// Mitsubishi GX Works2 project: PLC_Group22   PLC: FX3G

// global labels: Global1
VAR_GLOBAL
  START_DAY AT X007 : BOOL;
  EMERGENCY AT X005 : BOOL;
  DAY_IS_ON AT Y007 : BOOL;
  Input_Petel AT D2000 : REAL;
  Container_Petel AT D1100 : REAL;
  Input_Limon AT D2100 : REAL;
  Container_Limon AT D1200 : REAL;
  Input_Meyatzev AT D2200 : REAL;
  Container_Meyatzev AT D1300 : REAL;
  Input_Gumi AT D2300 : REAL;
  Container_Gumi AT D1400 : REAL;
  IceCream_Making AT X001 : BOOL;
  Gumigum_Type AT D8280 : INT;
  Chosen_Type AT D8202 : REAL;
END_VAR
VAR_GLOBAL CONSTANT
  Con_Value_6 : REAL := 6;
END_VAR
VAR_GLOBAL
  Regular AT M11 : BOOL;
  Pinuk AT M12 : BOOL;
  Enough_Petel_R AT M1 : BOOL;
  Enough_Limon_R AT M2 : BOOL;
  Enough_Meyatzev_R AT M3 : BOOL;
  Enough_Gumi_R AT M4 : BOOL;
  Enough_Regular AT M5 : BOOL;
END_VAR
VAR_GLOBAL CONSTANT
  Min_Petel_R : REAL := 280;
  Min_Limon_R : REAL := 455;
  Min_Meyatzev_R : REAL := 105;
  Min_Gumi_R : REAL := 28;
  Min_Petel_P : REAL := 385;
  Min_Limon_P : REAL := 665;
  Min_Meyatzev_P : REAL := 210;
  Min_Gumi_P : REAL := 70;
END_VAR
VAR_GLOBAL
  Enough_Petel_P AT M6 : BOOL;
  Enough_Limon_P AT M7 : BOOL;
  Enough_Meyatzev_P AT M8 : BOOL;
  Enough_Gumi_P AT M9 : BOOL;
  Enough_Pinuk AT M10 : BOOL;
END_VAR
VAR_GLOBAL CONSTANT
  Divv : REAL := 400;
  Sub280 : REAL := 280;
  Sub35 : REAL := 35;
  Sub420 : REAL := 420;
  Sub70 : REAL := 70;
  Timer5 : INT := 50;
END_VAR
VAR_GLOBAL
  IceCream_Making_Time AT TC1 : BOOL;
  StartMaking AT TS1 : BOOL;
  IsMakingIceCrem AT Y000 : BOOL;
END_VAR
VAR_GLOBAL CONSTANT
  Sub385 : REAL := 385;
  Sub105 : REAL := 105;
  Sub560 : REAL := 560;
  Sub140 : REAL := 140;
END_VAR
VAR_GLOBAL
  IceCream_Cooling AT X002 : BOOL;
END_VAR
VAR_GLOBAL CONSTANT
  Petel350 : REAL := 350;
END_VAR
VAR_GLOBAL
  CoolingPetel AT D1500 : REAL;
END_VAR
VAR_GLOBAL CONSTANT
  Limon490 : REAL := 490;
END_VAR
VAR_GLOBAL
  CoolingLimon AT D1600 : REAL;
  StartCooling AT TS2 : BOOL;
  Under10 AT X003 : BOOL;
  CoolingTimer AT TC2 : BOOL;
END_VAR
VAR_GLOBAL CONSTANT
  CoolingTime : INT := 80;
END_VAR
VAR_GLOBAL
  IsCoolingg AT Y002 : BOOL;
END_VAR
VAR_GLOBAL CONSTANT
  Petel560 : REAL := 560;
  Limon700 : REAL := 700;
END_VAR
VAR_GLOBAL
  End_Cooling_R AT M63 : BOOL;
  End_Cooling_P AT M64 : BOOL;
END_VAR
VAR_GLOBAL CONSTANT
  Cooling_Containers_R : REAL := 868;
  Gumi_R28 : REAL := 28;
END_VAR
VAR_GLOBAL
  Mixing_R_Timer AT TC3 : BOOL;
END_VAR
VAR_GLOBAL CONSTANT
  Mixing_R_Time : INT := 30;
END_VAR
VAR_GLOBAL
  Start_Mixing_R AT TS3 : BOOL;
  End_Mixing_R AT M65 : BOOL;
  Lights1 AT TC4 : BOOL;
END_VAR
VAR_GLOBAL CONSTANT
  Lights_Timer : INT := 5;
END_VAR
VAR_GLOBAL
  Lights1_on AT TS4 : BOOL;
  Lights1_Is_On AT Y005 : BOOL;
  Lights2 AT TC5 : BOOL;
  Lights2_on AT TS5 : BOOL;
  Lights2_Is_On AT Y006 : BOOL;
  Lights12 AT M66 : BOOL;
END_VAR
VAR_GLOBAL CONSTANT
  Cooling_Containers_P : REAL := 1330;
  Gumi_P70 : REAL := 70;
END_VAR
VAR_GLOBAL
  Mixing_P_Timer AT TC6 : BOOL;
END_VAR
VAR_GLOBAL CONSTANT
  Mixing_P_Time : INT := 50;
END_VAR
VAR_GLOBAL
  Start_Mixing_P AT TS6 : BOOL;
  End_Mixing_P AT M67 : BOOL;
  IceCream_Packing AT X004 : BOOL;
  Single_Unit_Packing AT X000 : BOOL;
  Units_Conter AT CC1 : BOOL;
END_VAR
VAR_GLOBAL CONSTANT
  Con_1 : REAL := 1;
END_VAR
VAR_GLOBAL
  Packages_Count AT D1900 : REAL;
  Counter_State AT CS1 : BOOL;
END_VAR
VAR_GLOBAL CONSTANT
  Min_1 : INT := 1;
  Value_7 : INT := 7;
END_VAR
VAR_GLOBAL
  Units AT CN1 : INT;
  In_Packing AT Y004 : BOOL;
  Mixing AT D1700 : REAL;
END_VAR
VAR_GLOBAL CONSTANT
  Sub124 : REAL := 124;
  Sub190 : REAL := 190;
  zero : REAL;
END_VAR
VAR_GLOBAL
  End_Packing AT M80 : BOOL;
  End_Of_The_Day AT M27 : BOOL;
  Output AT D8282 : INT;
END_VAR
VAR_GLOBAL CONSTANT
  Div40 : REAL := 40;
END_VAR
VAR_GLOBAL
  Not_Enough_Material AT M25 : BOOL;
END_VAR

// task Task_01 (event TRUE, interval 0, priority 31): POU_01

PROGRAM POU_01
(* structured ladder/FBD written out as ST: instructions are called as NAME(EN, inputs, outputs); _pN, _eN, _tN stand for wires *)
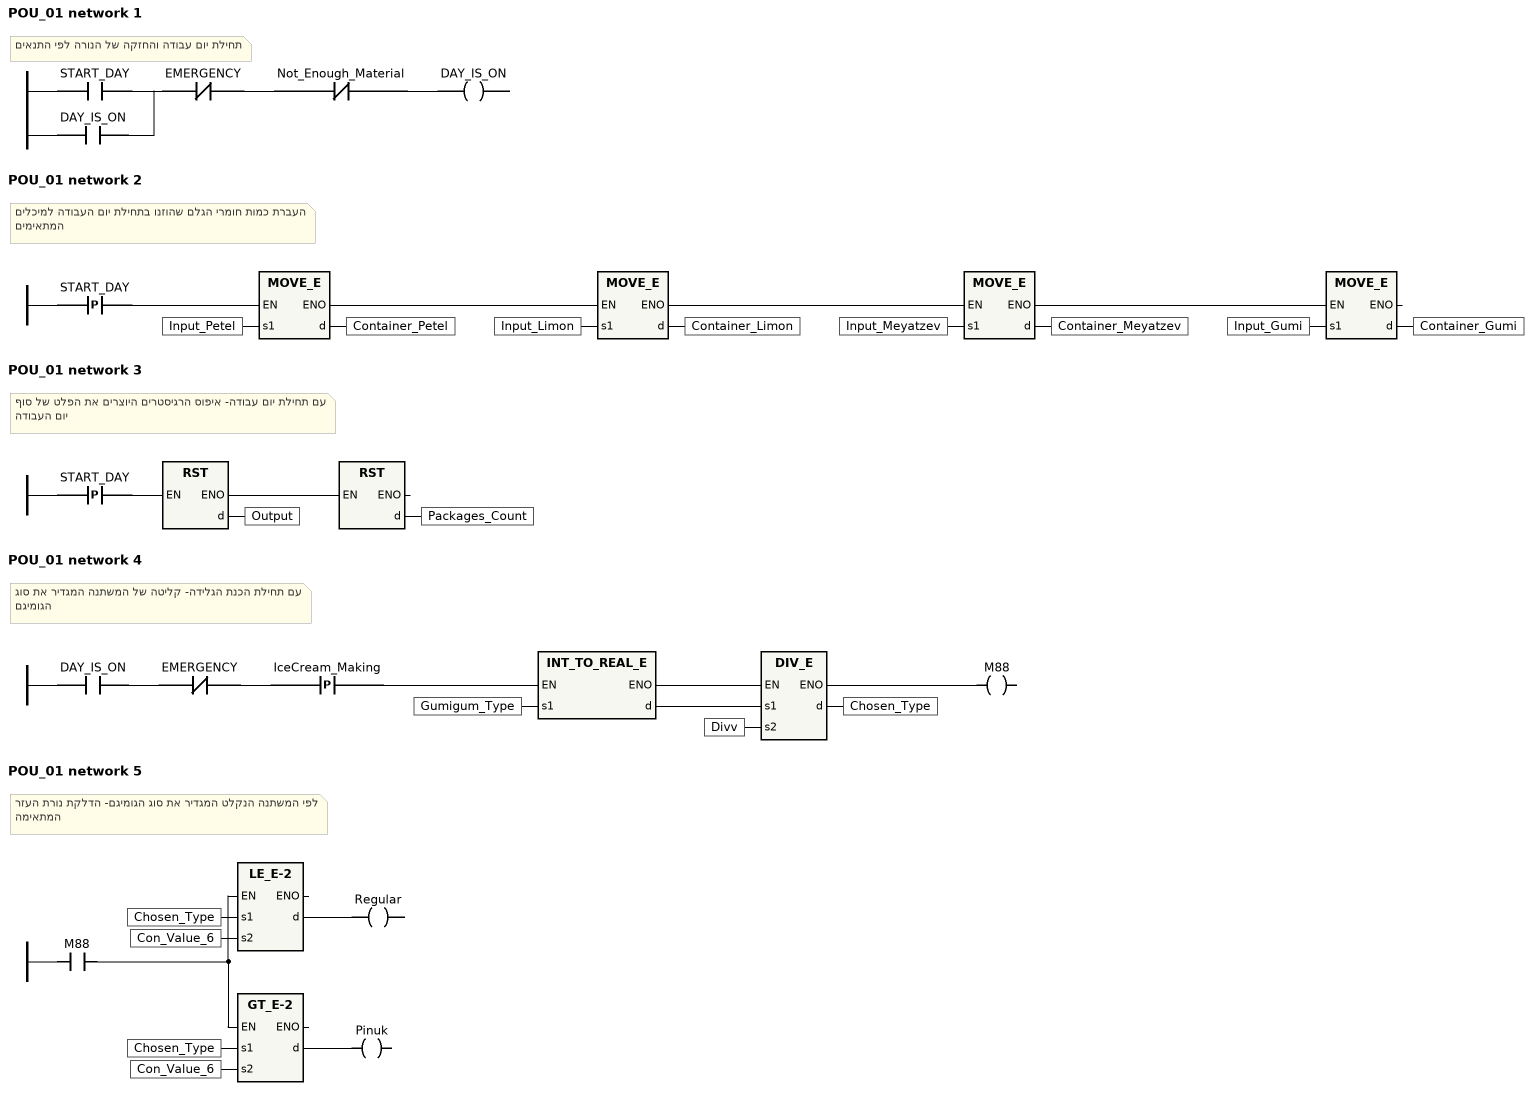
(* network 1 *)
(* תחילת יום עבודה והחזקה של הנורה לפי התנאים *)
DAY_IS_ON := ((START_DAY OR DAY_IS_ON) AND NOT EMERGENCY) AND NOT Not_Enough_Material;
(* network 2 *)
(* העברת כמות חומרי הגלם שהוזנו בתחילת יום העבודה למיכלים המתאימים *)
_e1 := MOVE_E(LDP(TRUE, START_DAY), Input_Petel, Container_Petel);
_e2 := MOVE_E(_e1, Input_Limon, Container_Limon);
_e3 := MOVE_E(_e2, Input_Meyatzev, Container_Meyatzev);
MOVE_E(_e3, Input_Gumi, Container_Gumi);
(* network 3 *)
(* עם תחילת יום עבודה- איפוס הרגיסטרים היוצרים את הפלט של סוף יום העבודה *)
_e1 := RST(LDP(TRUE, START_DAY), Output);
RST(_e1, Packages_Count);
(* network 4 *)
(* עם תחילת הכנת הגלידה- קליטה של המשתנה המגדיר את סוג הגומיגם *)
_e2 := INT_TO_REAL_E(DAY_IS_ON AND NOT EMERGENCY AND LDP(TRUE, IceCream_Making), Gumigum_Type, _t1);
_e3 := DIV_E(_e2, _t1, Divv, Chosen_Type);
M88 := _e3;
(* network 5 *)
(* לפי המשתנה הנקלט המגדיר את סוג הגומיגם- הדלקת נורת העזר המתאימה *)
LE_E(M88, Chosen_Type, Con_Value_6, _t1);
Regular := _t1;
GT_E(M88, Chosen_Type, Con_Value_6, _t2);
Pinuk := _t2;
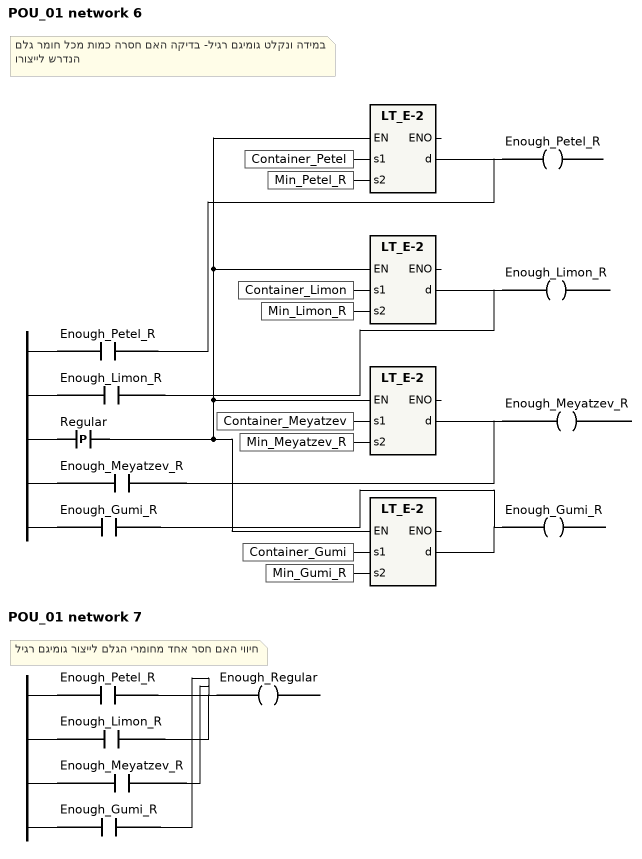
(* network 6 *)
(* במידה ונקלט גומיגם רגיל- בדיקה האם חסרה כמות מכל חומר גלם הנדרש לייצורו *)
_p1 := LDP(TRUE, Regular);
LT_E(_p1, Container_Petel, Min_Petel_R, _t2);
Enough_Petel_R := Enough_Petel_R OR _t2;
LT_E(_p1, Container_Limon, Min_Limon_R, _t3);
Enough_Limon_R := Enough_Limon_R OR _t3;
LT_E(_p1, Container_Meyatzev, Min_Meyatzev_R, _t4);
Enough_Meyatzev_R := _t4 OR Enough_Meyatzev_R;
LT_E(_p1, Container_Gumi, Min_Gumi_R, _t5);
Enough_Gumi_R := _t5 OR Enough_Gumi_R;
(* network 7 *)
(* חיווי האם חסר אחד מחומרי הגלם לייצור גומיגם רגיל *)
Enough_Regular := Enough_Petel_R OR Enough_Limon_R OR Enough_Meyatzev_R OR Enough_Gumi_R;
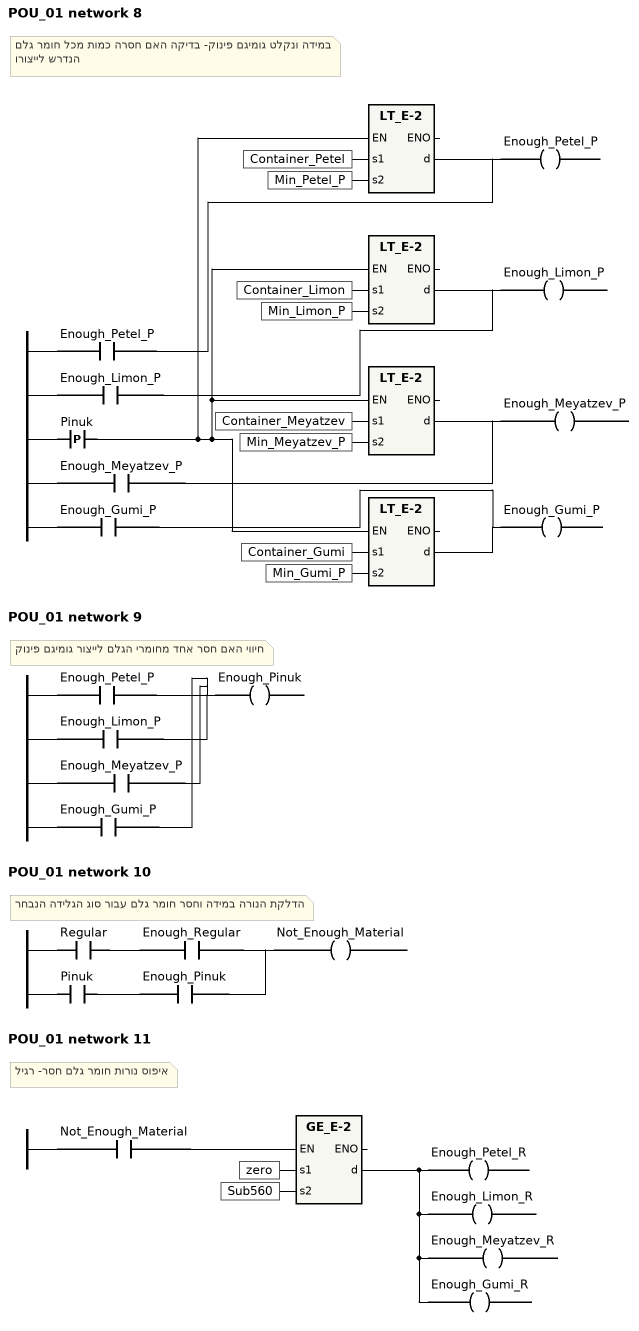
(* network 8 *)
(* במידה ונקלט גומיגם פינוק- בדיקה האם חסרה כמות מכל חומר גלם הנדרש לייצורו *)
_p1 := LDP(TRUE, Pinuk);
LT_E(_p1, Container_Petel, Min_Petel_P, _t2);
Enough_Petel_P := Enough_Petel_P OR _t2;
LT_E(_p1, Container_Limon, Min_Limon_P, _t3);
Enough_Limon_P := Enough_Limon_P OR _t3;
LT_E(_p1, Container_Meyatzev, Min_Meyatzev_P, _t4);
Enough_Meyatzev_P := _t4 OR Enough_Meyatzev_P;
LT_E(_p1, Container_Gumi, Min_Gumi_P, _t5);
Enough_Gumi_P := _t5 OR Enough_Gumi_P;
(* network 9 *)
(* חיווי האם חסר אחד מחומרי הגלם לייצור גומיגם פינוק *)
Enough_Pinuk := Enough_Petel_P OR Enough_Limon_P OR Enough_Meyatzev_P OR Enough_Gumi_P;
(* network 10 *)
(* הדלקת הנורה במידה וחסר חומר גלם עבור סוג הגלידה הנבחר *)
Not_Enough_Material := (Regular AND Enough_Regular) OR (Pinuk AND Enough_Pinuk);
(* network 11 *)
(* איפוס נורות חומר גלם חסר- רגיל *)
GE_E(Not_Enough_Material, zero, Sub560, _t1);
Enough_Petel_R := _t1;
Enough_Limon_R := _t1;
Enough_Meyatzev_R := _t1;
Enough_Gumi_R := _t1;
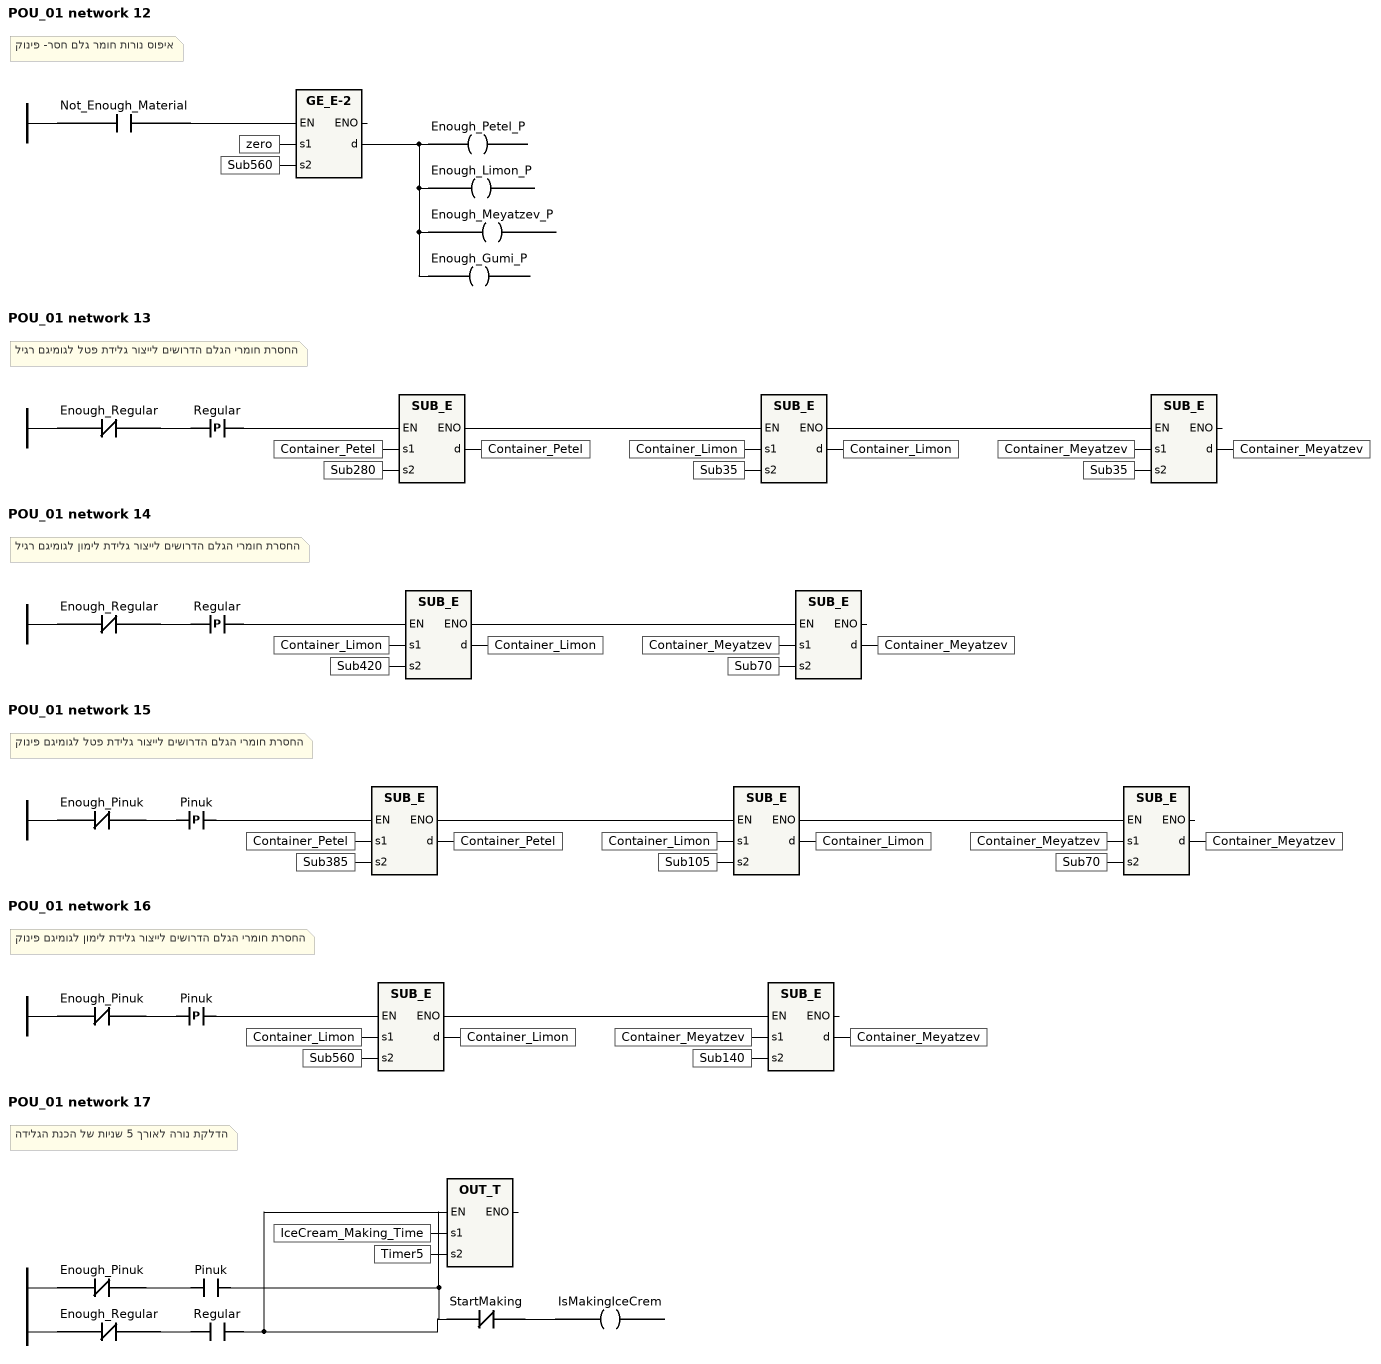
(* network 12 *)
(* איפוס נורות חומר גלם חסר- פינוק *)
GE_E(Not_Enough_Material, zero, Sub560, _t1);
Enough_Petel_P := _t1;
Enough_Limon_P := _t1;
Enough_Meyatzev_P := _t1;
Enough_Gumi_P := _t1;
(* network 13 *)
(* החסרת חומרי הגלם הדרושים לייצור גלידת פטל לגומיגם רגיל *)
_e1 := SUB_E(NOT Enough_Regular AND LDP(TRUE, Regular), Container_Petel, Sub280, Container_Petel);
_e2 := SUB_E(_e1, Container_Limon, Sub35, Container_Limon);
SUB_E(_e2, Container_Meyatzev, Sub35, Container_Meyatzev);
(* network 14 *)
(* החסרת חומרי הגלם הדרושים לייצור גלידת לימון לגומיגם רגיל *)
_e1 := SUB_E(NOT Enough_Regular AND LDP(TRUE, Regular), Container_Limon, Sub420, Container_Limon);
SUB_E(_e1, Container_Meyatzev, Sub70, Container_Meyatzev);
(* network 15 *)
(* החסרת חומרי הגלם הדרושים לייצור גלידת פטל לגומיגם פינוק *)
_e1 := SUB_E(NOT Enough_Pinuk AND LDP(TRUE, Pinuk), Container_Petel, Sub385, Container_Petel);
_e2 := SUB_E(_e1, Container_Limon, Sub105, Container_Limon);
SUB_E(_e2, Container_Meyatzev, Sub70, Container_Meyatzev);
(* network 16 *)
(* החסרת חומרי הגלם הדרושים לייצור גלידת לימון לגומיגם פינוק *)
_e1 := SUB_E(NOT Enough_Pinuk AND LDP(TRUE, Pinuk), Container_Limon, Sub560, Container_Limon);
SUB_E(_e1, Container_Meyatzev, Sub140, Container_Meyatzev);
(* network 17 *)
(* הדלקת נורה לאורך 5 שניות של הכנת הגלידה *)
_p1 := (NOT Enough_Pinuk AND Pinuk) OR (NOT Enough_Regular AND Regular);
OUT_T(_p1, IceCream_Making_Time, Timer5);
IsMakingIceCrem := _p1 AND NOT StartMaking;
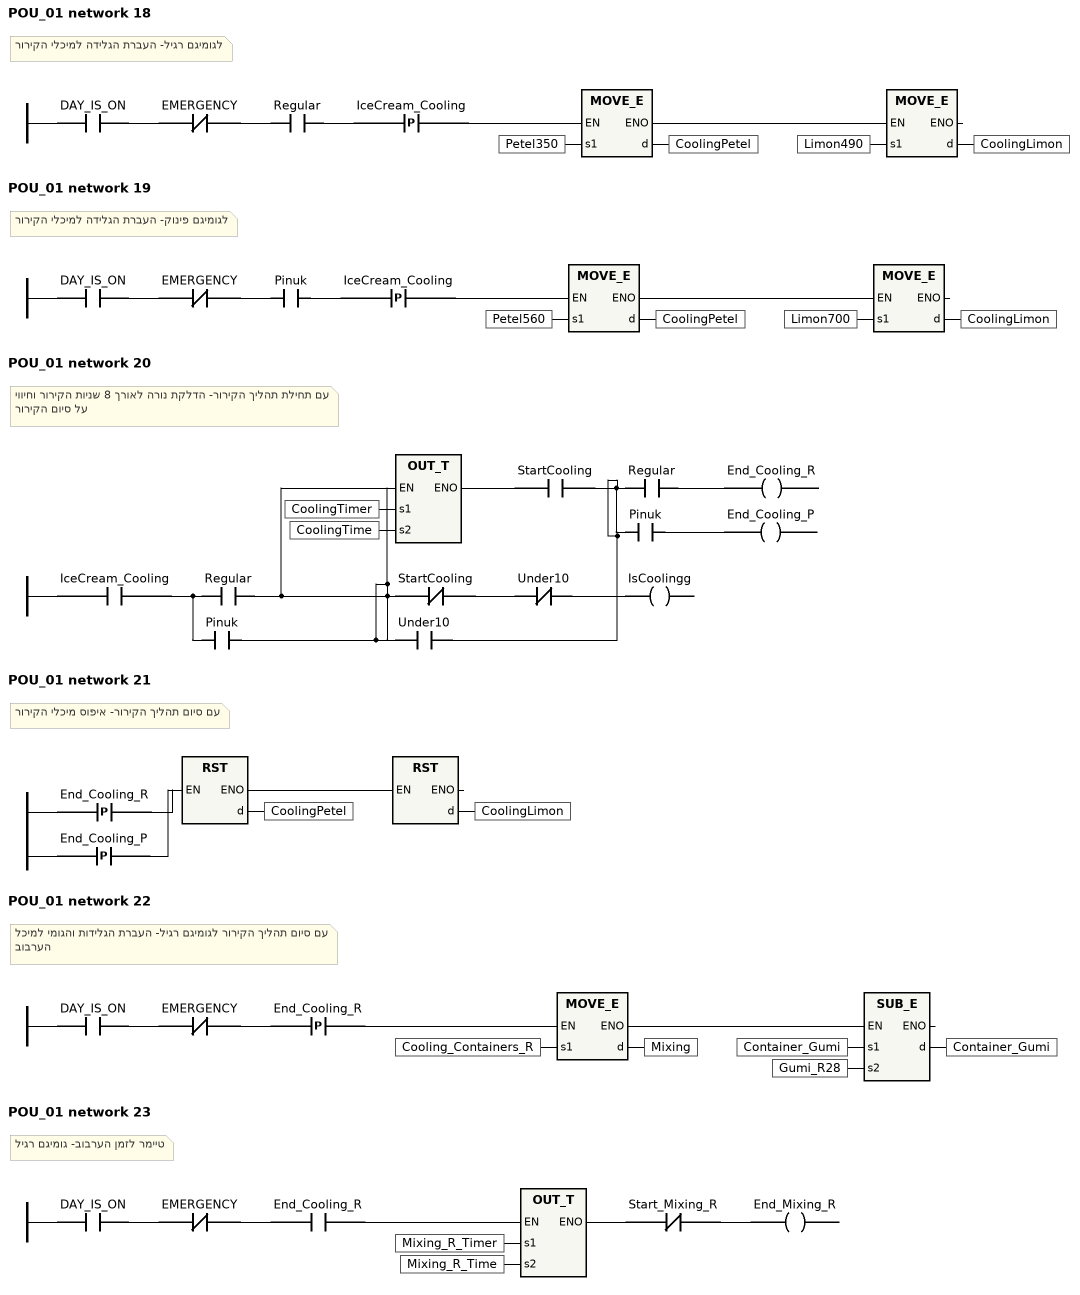
(* network 18 *)
(* לגומיגם רגיל- העברת הגלידה למיכלי הקירור *)
_e1 := MOVE_E(DAY_IS_ON AND NOT EMERGENCY AND Regular AND LDP(TRUE, IceCream_Cooling), Petel350, CoolingPetel);
MOVE_E(_e1, Limon490, CoolingLimon);
(* network 19 *)
(* לגומיגם פינוק- העברת הגלידה למיכלי הקירור *)
_e1 := MOVE_E(DAY_IS_ON AND NOT EMERGENCY AND Pinuk AND LDP(TRUE, IceCream_Cooling), Petel560, CoolingPetel);
MOVE_E(_e1, Limon700, CoolingLimon);
(* network 20 *)
(* עם תחילת תהליך הקירור- הדלקת נורה לאורך 8 שניות הקירור וחיווי על סיום הקירור *)
_p1 := (IceCream_Cooling AND Regular) OR (IceCream_Cooling AND Pinuk);
_e2 := OUT_T(_p1, CoolingTimer, CoolingTime);
_p3 := (_e2 AND StartCooling) OR (_p1 AND Under10);
End_Cooling_R := _p3 AND Regular;
End_Cooling_P := _p3 AND Pinuk;
IsCoolingg := _p1 AND NOT StartCooling AND NOT Under10;
(* network 21 *)
(* עם סיום תהליך הקירור- איפוס מיכלי הקירור *)
_e1 := RST(LDP(TRUE, End_Cooling_R) OR LDP(TRUE, End_Cooling_P), CoolingPetel);
RST(_e1, CoolingLimon);
(* network 22 *)
(* עם סיום תהליך הקירור לגומיגם רגיל- העברת הגלידות והגומי למיכל הערבוב *)
_e1 := MOVE_E(DAY_IS_ON AND NOT EMERGENCY AND LDP(TRUE, End_Cooling_R), Cooling_Containers_R, Mixing);
SUB_E(_e1, Container_Gumi, Gumi_R28, Container_Gumi);
(* network 23 *)
(* טיימר לזמן הערבוב- גומיגם רגיל *)
_e1 := OUT_T(DAY_IS_ON AND NOT EMERGENCY AND End_Cooling_R, Mixing_R_Timer, Mixing_R_Time);
End_Mixing_R := _e1 AND NOT Start_Mixing_R;
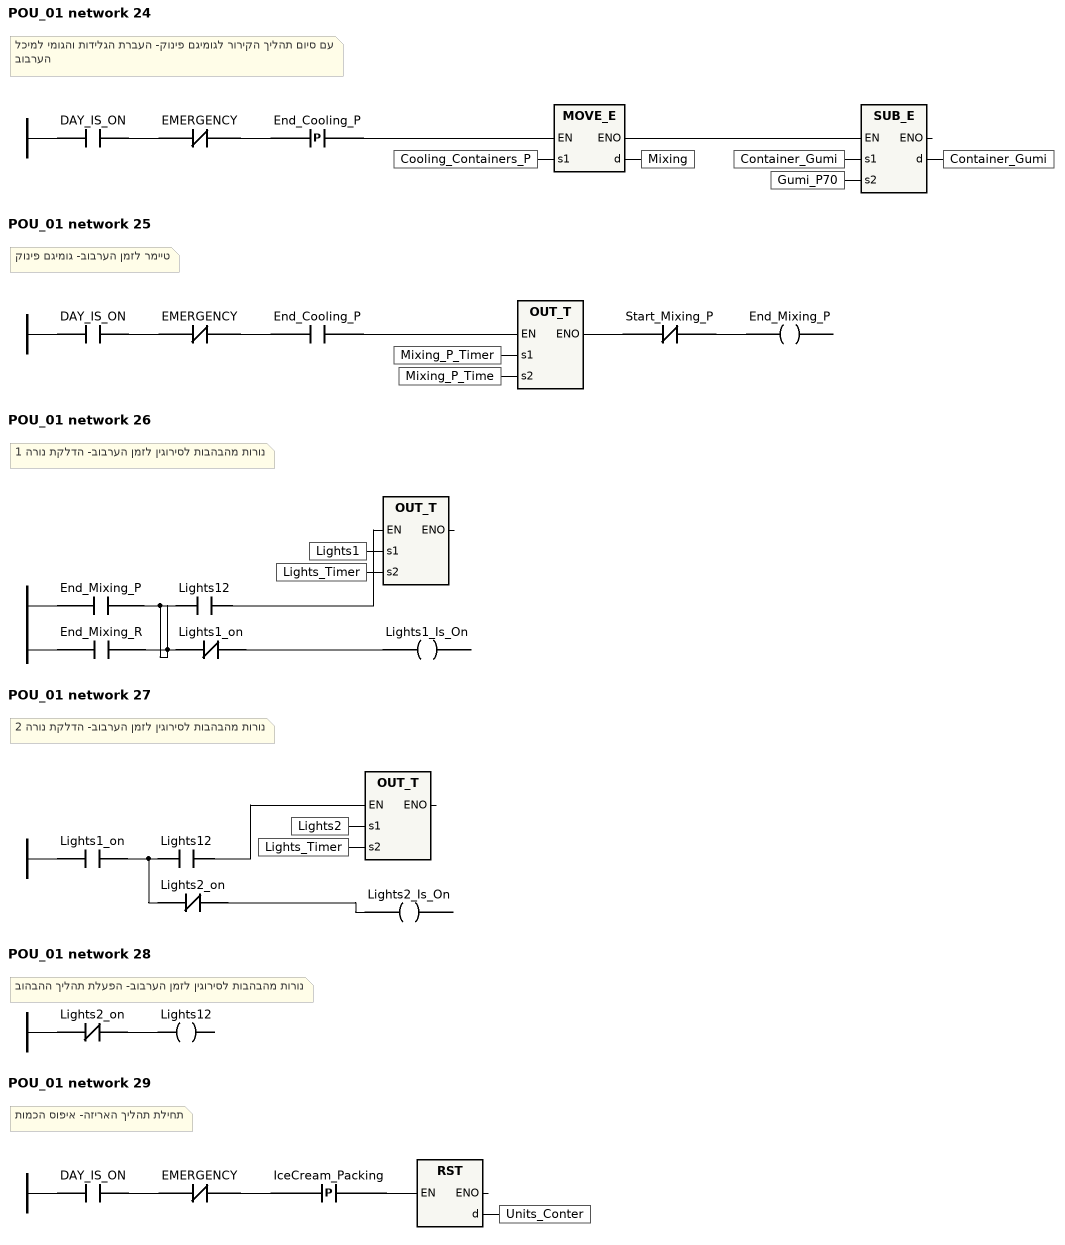
(* network 24 *)
(* עם סיום תהליך הקירור לגומיגם פינוק- העברת הגלידות והגומי למיכל הערבוב *)
_e1 := MOVE_E(DAY_IS_ON AND NOT EMERGENCY AND LDP(TRUE, End_Cooling_P), Cooling_Containers_P, Mixing);
SUB_E(_e1, Container_Gumi, Gumi_P70, Container_Gumi);
(* network 25 *)
(* טיימר לזמן הערבוב- גומיגם פינוק *)
_e1 := OUT_T(DAY_IS_ON AND NOT EMERGENCY AND End_Cooling_P, Mixing_P_Timer, Mixing_P_Time);
End_Mixing_P := _e1 AND NOT Start_Mixing_P;
(* network 26 *)
(* נורות מהבהבות לסירוגין לזמן הערבוב- הדלקת נורה 1 *)
_p1 := End_Mixing_P OR End_Mixing_R;
OUT_T(_p1 AND Lights12, Lights1, Lights_Timer);
Lights1_Is_On := _p1 AND NOT Lights1_on;
(* network 27 *)
(* נורות מהבהבות לסירוגין לזמן הערבוב- הדלקת נורה 2 *)
OUT_T(Lights1_on AND Lights12, Lights2, Lights_Timer);
Lights2_Is_On := Lights1_on AND NOT Lights2_on;
(* network 28 *)
(* נורות מהבהבות לסירוגין לזמן הערבוב- הפעלת תהליך ההבהוב *)
Lights12 := NOT Lights2_on;
(* network 29 *)
(* תחילת תהליך האריזה- איפוס הכמות *)
RST(DAY_IS_ON AND NOT EMERGENCY AND LDP(TRUE, IceCream_Packing), Units_Conter);
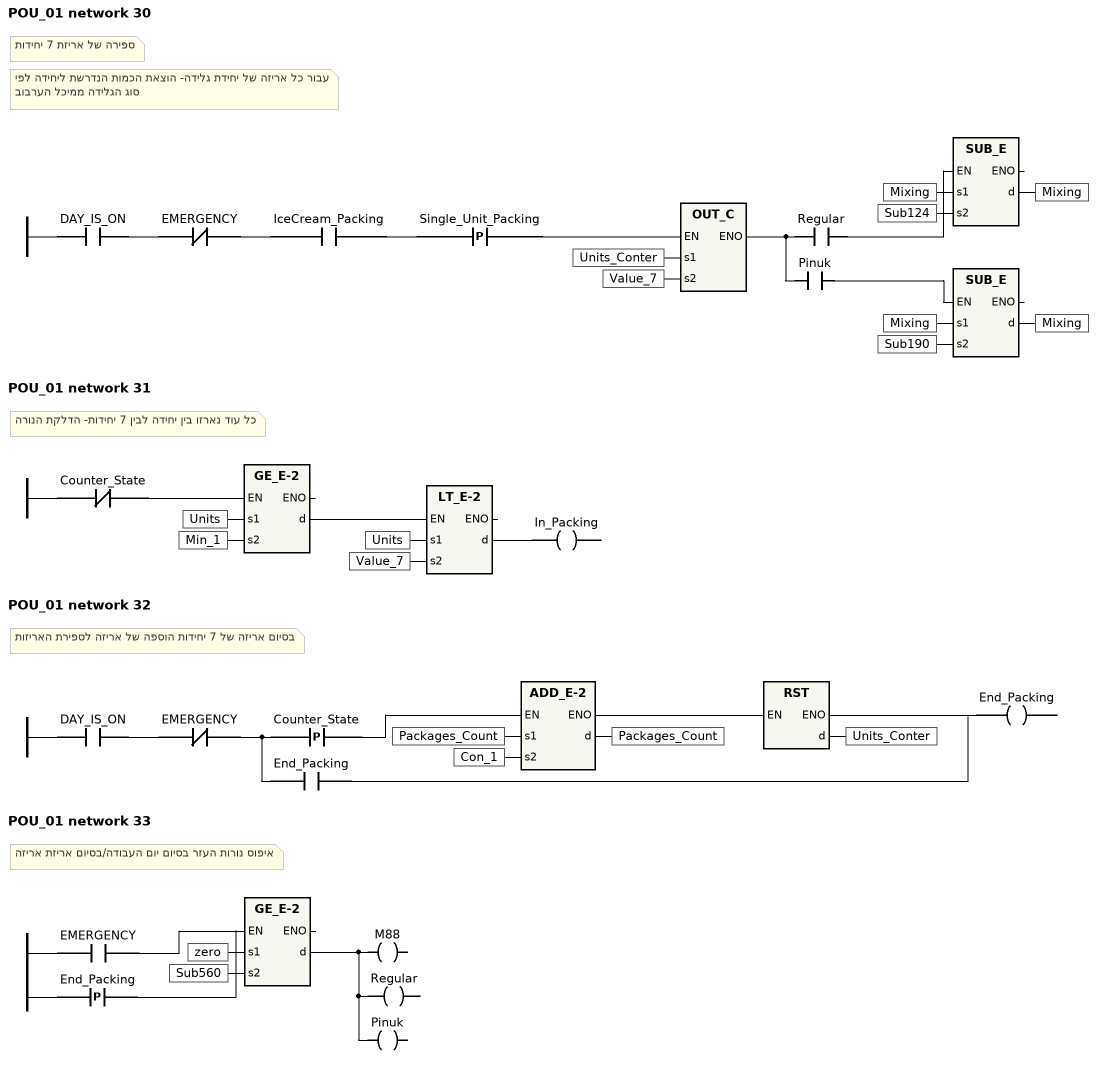
(* network 30 *)
(* ספירה של אריזת 7 יחידות *)
(* עבור כל אריזה של יחידת גלידה- הוצאת הכמות הנדרשת ליחידה לפי סוג הגלידה ממיכל הערבוב *)
_e1 := OUT_C(DAY_IS_ON AND NOT EMERGENCY AND IceCream_Packing AND LDP(TRUE, Single_Unit_Packing), Units_Conter, Value_7);
SUB_E(_e1 AND Regular, Mixing, Sub124, Mixing);
SUB_E(_e1 AND Pinuk, Mixing, Sub190, Mixing);
(* network 31 *)
(* כל עוד נארזו בין יחידה לבין 7 יחידות- הדלקת הנורה *)
GE_E(NOT Counter_State, Units, Min_1, _t1);
LT_E(_t1, Units, Value_7, _t2);
In_Packing := _t2;
(* network 32 *)
(* בסיום אריזה של 7 יחידות הוספה של אריזה לספירת האריזות *)
_p1 := DAY_IS_ON AND NOT EMERGENCY;
_e2 := ADD_E(_p1 AND LDP(TRUE, Counter_State), Packages_Count, Con_1, Packages_Count);
_e3 := RST(_e2, Units_Conter);
End_Packing := _e3 OR (_p1 AND End_Packing);
(* network 33 *)
(* איפוס נורות העזר בסיום יום העבודה/בסיום אריזת אריזה *)
GE_E(EMERGENCY OR LDP(TRUE, End_Packing), zero, Sub560, _t1);
M88 := _t1;
Regular := _t1;
Pinuk := _t1;
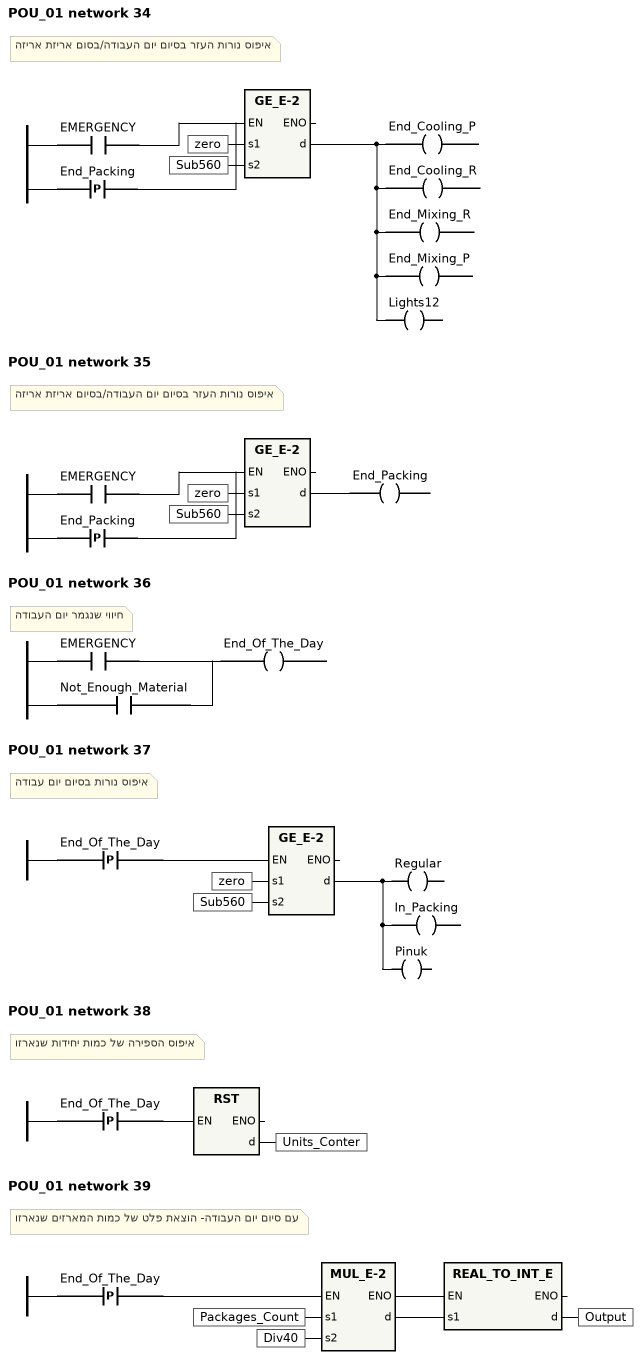
(* network 34 *)
(* איפוס נורות העזר בסיום יום העבודה/בסום אריזת אריזה *)
GE_E(EMERGENCY OR LDP(TRUE, End_Packing), zero, Sub560, _t1);
End_Cooling_P := _t1;
End_Cooling_R := _t1;
End_Mixing_R := _t1;
End_Mixing_P := _t1;
Lights12 := _t1;
(* network 35 *)
(* איפוס נורות העזר בסיום יום העבודה/בסיום אריזת אריזה *)
GE_E(EMERGENCY OR LDP(TRUE, End_Packing), zero, Sub560, _t1);
End_Packing := _t1;
(* network 36 *)
(* חיווי שנגמר יום העבודה *)
End_Of_The_Day := EMERGENCY OR Not_Enough_Material;
(* network 37 *)
(* איפוס נורות בסיום יום עבודה *)
GE_E(LDP(TRUE, End_Of_The_Day), zero, Sub560, _t1);
Regular := _t1;
In_Packing := _t1;
Pinuk := _t1;
(* network 38 *)
(* איפוס הספירה של כמות יחידות שנארזו *)
RST(LDP(TRUE, End_Of_The_Day), Units_Conter);
(* network 39 *)
(* עם סיום יום העבודה- הוצאת פלט של כמות המארזים שנארזו *)
_e2 := MUL_E(LDP(TRUE, End_Of_The_Day), Packages_Count, Div40, _t1);
REAL_TO_INT_E(_e2, _t1, Output);
END_PROGRAM
